// TIA Portal project "test" (V17)

(* hardware
DEVICE "S7-1500/ET200MP station_1"  S7-1500 station
   slot 0: "Rail_0"  Rack  6ES7 590-1***0-0AA0
   slot 1: "PLC_1"  CPU 1516-3 PN/DP  6ES7 516-3AN02-0AB0  V2.9
      slot 3: "CPU display_1"  6ES7591-1BA00-0AA0
      slot 32768: "PROFINET interface_1"  X1
      slot 33024: "PROFINET interface_2"  X2
      slot 33280: "DP interface_1"  X3
      slot 34817: "Virtual CP interface port_1"  Virtual CP interface port  Virtual CP interface port
DEVICE "S7-1500/ET200MP station_2"  S7-1500 station
   slot 0: "Rail_0"  Rack  6ES7 590-1***0-0AA0
   slot 1: "io device_1"  IM 155-5 PN HF  6ES7 155-5AA00-0AC0  V3.0
   slot 2: "DQ 32x24VDC/0.5A ST_1"  DQ 32x24VDC/0.5A ST  6ES7 522-1BL00-0AB0  V2.0
   slot 3: "AI 8xU/I/RTD/TC ST_1"  AI 8xU/I/RTD/TC ST  6ES7 531-7KF00-0AB0  V2.0
   slot 4: "AQ 4xU/I ST_1"  AQ 4xU/I ST  6ES7 532-5HD00-0AB0  V2.0
DEVICE "GSD device_1"  GSD.Device.PN
   slot 0: "Rack"  Rack  V1.0
   slot 0: "al1102_3"  AL1102  AL1102
      slot 0: "AL1102"  AL1102
      slot 1: "X1"  X1
         slot 1: "Port 1"  Port 1
         slot 2: "Port 2"  Port 2
      slot 1: "8 Ports_1"  8 Ports  AL1102
         slot 0: "IO-Link Master"  IO-Link Master
DEVICE "GSD device_2"  GSD.Device.PN
   slot 0: "Rack"  Rack  V1.0
   slot 0: "al1102_4"  AL1102  AL1102
      slot 0: "AL1102"  AL1102
      slot 1: "X1"  X1
         slot 1: "Port 1"  Port 1
         slot 2: "Port 2"  Port 2
      slot 1: "8 Ports_1"  8 Ports  AL1102
         slot 0: "IO-Link Master"  IO-Link Master
   slot 3: "IO-Link In  2 Byte + PQI"  IO-Link In  2 Byte + PQI
   slot 5: "IO-Link In  2 Byte + PQI_1"  IO-Link In  2 Byte + PQI
   slot 6: "IO-Link In  8 Byte + PQI"  IO-Link In  8 Byte + PQI
   slot 7: "IO-Link In  2 Byte + PQI_2"  IO-Link In  2 Byte + PQI
   slot 8: "IO-Link In  2 Byte + PQI_3"  IO-Link In  2 Byte + PQI
DEVICE "GSD device_3"  GSD.Device.PN
   slot 0: "Rack"  Rack  V1.0
   slot 0: "al1102_2"  AL1102  AL1102
      slot 0: "AL1102"  AL1102
      slot 1: "X1"  X1
         slot 1: "Port 1"  Port 1
         slot 2: "Port 2"  Port 2
      slot 1: "8 Ports_1"  8 Ports  AL1102
         slot 0: "IO-Link Master"  IO-Link Master
*)

// ===== PLC "PLC_1"  CPU 1516-3 PN/DP =====

VAR_GLOBAL   // PLC tag table "Default tag table"
   "firstHeater" AT %Q0.5 : Bool;
   "secondHeater" AT %Q0.6 : Bool;
   "thirdHeater" AT %Q0.7 : Bool;
   "tempAfter" AT %IW8 : Int;
   "tempBefore" AT %IW14 : Int;
   "valve" AT %QW8 : Int;
   "flowFlow" AT %IW32 : Int;
   "power" AT %MD50 : Real;
   "flowTemp" AT %IW34 : Int;
   "Tag_1" AT %M100.0 : Bool;
END_VAR

TYPE "UDT_Pomiar"
VERSION : 0.1
   STRUCT
      power : UDInt;
      switchesFirst : UDInt;
      switchesSecond : UDInt;
      switchesThird : UDInt;
      onePhase : UDInt;
      threePhase : UDInt;
   END_STRUCT;
END_TYPE

DATA_BLOCK "ExecutePWM_DB"   // DB1
{ S7_Optimized_Access := 'TRUE' }
VERSION : 0.1
// stored: InstanceOfName ExecutePWM
"ExecutePWM"
BEGIN
END_DATA_BLOCK

DATA_BLOCK "Analysis_DB"   // DB2
{ S7_Optimized_Access := 'TRUE' }
VERSION : 0.1
// stored: InstanceOfName Analysis
"Analysis"
BEGIN
END_DATA_BLOCK

// folder: System blocks/Program resources

DATA_BLOCK "IEC_Timer_0_DB_2"   // DB3
{ S7_Optimized_Access := 'TRUE' }
AUTHOR : Simatic
FAMILY : IEC
NAME : IEC_TMR
VERSION : 1.0
// stored: InstanceOfName IEC_TIMER
"IEC_TIMER"
BEGIN
END_DATA_BLOCK

DATA_BLOCK "IEC_Timer_0_DB_1"   // DB4
{ S7_Optimized_Access := 'TRUE' }
AUTHOR : Simatic
FAMILY : IEC
NAME : IEC_TMR
VERSION : 1.0
// stored: InstanceOfName IEC_TIMER
"IEC_TIMER"
BEGIN
END_DATA_BLOCK

// folder: (top level)

FUNCTION_BLOCK "ControlPWM"   // FB1, LAD
TITLE = ControlPWM
{ S7_Optimized_Access := 'TRUE' }
VERSION : 0.1
// Obsługa wypełnienia dla każdej z grzałek, w zależności od wyboru trybu pracy (jednofazowy lub trójfazowy).
   VAR_INPUT
      I_cycleTime : DInt;   // given in milliseconds
      I_filling_1 : Int;   // <0, 100>
      I_filling_2 : Int;   // <0, 100>
      I_filling_3 : Int;   // <0, 100>
      I_OnePhaseSwitch : Bool;
      I_threePhaseSwitch : Bool;
   END_VAR
   VAR_OUTPUT
      O_heaterState_1 : Bool;
      O_heaterState_2 : Bool;
      O_heaterState_3 : Bool;
   END_VAR
   VAR
      IEC_Timer_11 : TON_TIME;
      IEC_Timer_12 : TON_TIME;
      highStateNum_1 : DInt;   // given in milliseconds
      lowStateNum_1 : DInt;   // given in milliseconds
      highStateTime_1 : Time;   // given in milliseconds
      lowStateTime_1 : Time;   // given in milliseconds
      IEC_Timer_21 : TON_TIME;
      IEC_Timer_22 : TON_TIME;
      highStateNum_2 : DInt;   // given in milliseconds
      lowStateNum_2 : DInt;   // given in milliseconds
      highStateTime_2 : Time;   // given in milliseconds
      lowStateTime_2 : Time;   // given in milliseconds
      IEC_Timer_31 : TON_TIME;
      IEC_Timer_32 : TON_TIME;
      highStateNum_3 : DInt;   // given in milliseconds
      lowStateNum_3 : DInt;   // given in milliseconds
      highStateTime_3 : Time;   // given in milliseconds
      lowStateTime_3 : Time;   // given in milliseconds
      IEC_Timer_0_Instance : TON_TIME;
      IEC_Timer_0_Instance_1 : TON_TIME;
   END_VAR
BEGIN

REGION Network 1: Obliczenie czasu stanów
   // Blok calculate oblicza czas na podstawie wartości procentowej (I_filling_X) i przypisuje wartości czasowe stanu wysokiego oraz niskiego (Int) do odpowiednich zmiennych (highStateNum_X, lowStateNum_X).
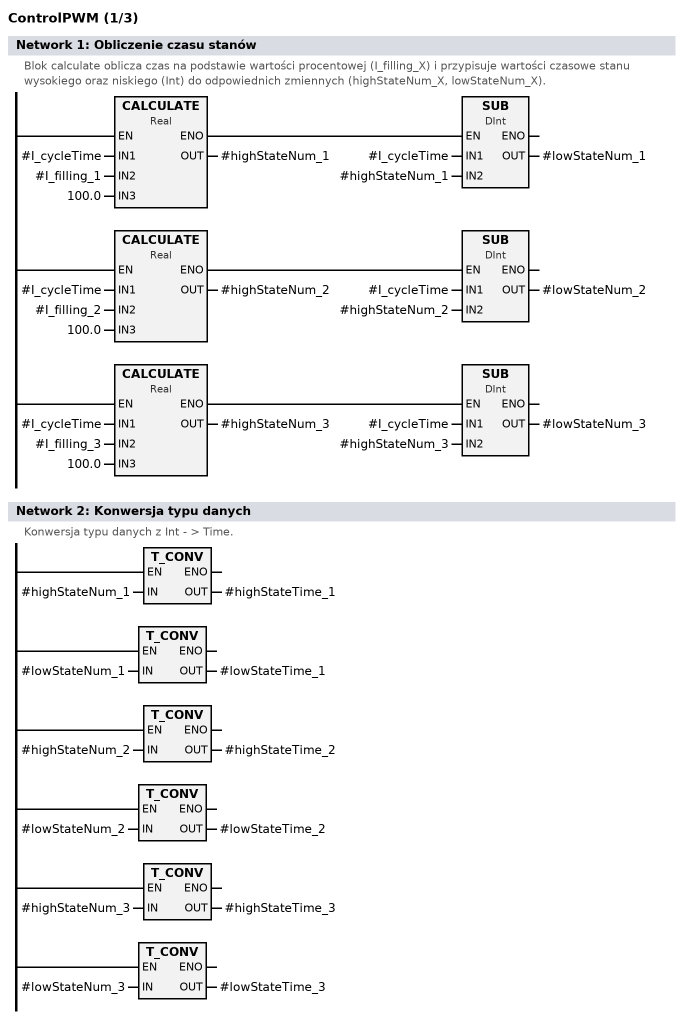
   RUNG wire#powerrail
      { S7_Templates := "SrcType := Real"; S7_Expression := "(IN1*IN2)/IN3" } Calculate(in1 := #I_cycleTime, in2 := #I_filling_1, in3 := 100.0, out => #highStateNum_1)
      { S7_Templates := "SrcType := DInt" } Sub(in1 := #I_cycleTime, in2 := #highStateNum_1, out => #lowStateNum_1)
   END_RUNG
   RUNG wire#powerrail
      { S7_Templates := "SrcType := Real"; S7_Expression := "(IN1*IN2)/IN3" } Calculate(in1 := #I_cycleTime, in2 := #I_filling_2, in3 := 100.0, out => #highStateNum_2)
      { S7_Templates := "SrcType := DInt" } Sub(in1 := #I_cycleTime, in2 := #highStateNum_2, out => #lowStateNum_2)
   END_RUNG
   RUNG wire#powerrail
      { S7_Templates := "SrcType := Real"; S7_Expression := "(IN1*IN2)/IN3" } Calculate(in1 := #I_cycleTime, in2 := #I_filling_3, in3 := 100.0, out => #highStateNum_3)
      { S7_Templates := "SrcType := DInt" } Sub(in1 := #I_cycleTime, in2 := #highStateNum_3, out => #lowStateNum_3)
   END_RUNG
   // the same network as SCL:
   #highStateNum_1 := (#I_cycleTime*#I_filling_1)/100.0;
   #lowStateNum_1 := #I_cycleTime - #highStateNum_1;
   #highStateNum_2 := (#I_cycleTime*#I_filling_2)/100.0;
   #lowStateNum_2 := #I_cycleTime - #highStateNum_2;
   #highStateNum_3 := (#I_cycleTime*#I_filling_3)/100.0;
   #lowStateNum_3 := #I_cycleTime - #highStateNum_3;
END_REGION

REGION Network 2: Konwersja typu danych
   // Konwersja typu danych z Int - > Time.
   #highStateTime_1 := T_CONV(IN := #highStateNum_1);
   #lowStateTime_1 := T_CONV(IN := #lowStateNum_1);
   #highStateTime_2 := T_CONV(IN := #highStateNum_2);
   #lowStateTime_2 := T_CONV(IN := #lowStateNum_2);
   #highStateTime_3 := T_CONV(IN := #highStateNum_3);
   #lowStateTime_3 := T_CONV(IN := #lowStateNum_3);
END_REGION

REGION Network 3: Kontrola wypełnienia trybu trójfazowego (1)
   // Wypełnienie jest kontrolowane na podstawie dwóch zegarów TON. Każdy ze stanów uruchamia zegar, który odlicza czas (opóźninie) do uruchomienia stanu przeciwnego. Timery działają na przemian i nie mogą zostac uruchomione jednocześnie. Po zmianie stanu, licznik stanu przeciwnego zostaje zresetowany zgodnie z działaniem zegara TON. Logika ta działa nieprawidłowo, gdy któryś z określonych czasów jest równy 0, stąd dwie ostatnie gałęzie usprawniające działanie.
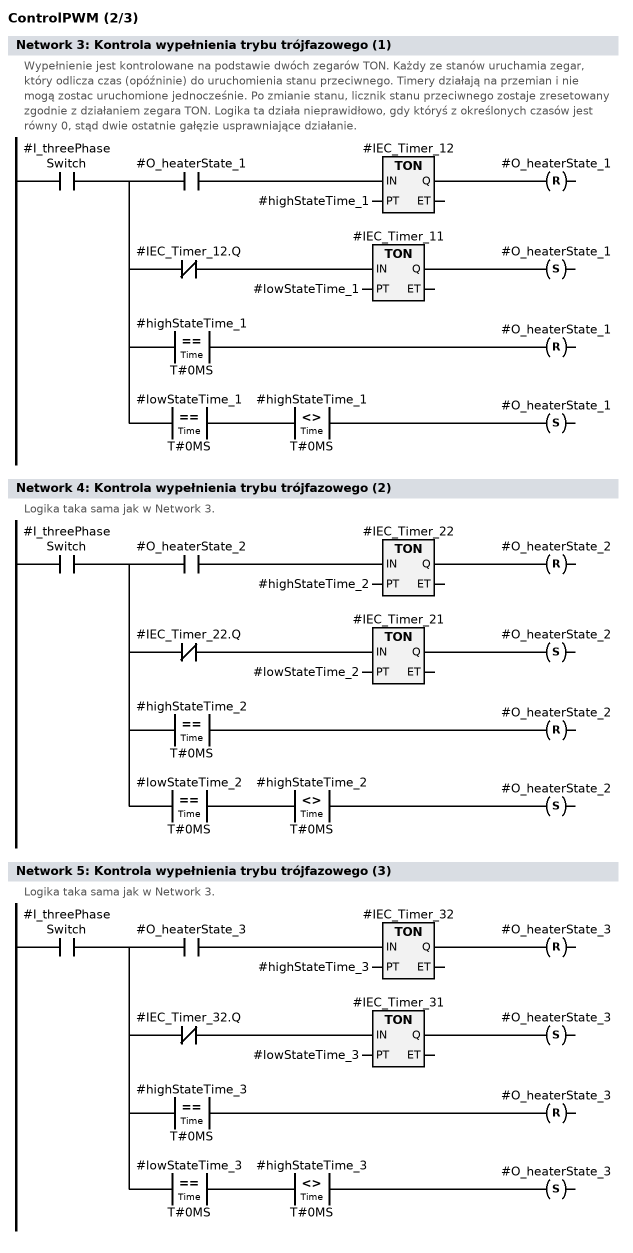
   #IEC_Timer_12(IN := #I_threePhaseSwitch AND #O_heaterState_1, PT := #highStateTime_1);   // TON
   IF #IEC_Timer_12.Q THEN #O_heaterState_1 := FALSE; END_IF;
   #IEC_Timer_11(IN := #I_threePhaseSwitch AND NOT #IEC_Timer_12.Q, PT := #lowStateTime_1);   // TON
   IF #IEC_Timer_11.Q THEN #O_heaterState_1 := TRUE; END_IF;
   IF #I_threePhaseSwitch AND (#highStateTime_1 = T#0MS) THEN #O_heaterState_1 := FALSE; END_IF;
   IF #I_threePhaseSwitch AND (#lowStateTime_1 = T#0MS) AND (#highStateTime_1 <> T#0MS) THEN
       #O_heaterState_1 := TRUE;
   END_IF;
END_REGION

REGION Network 4: Kontrola wypełnienia trybu trójfazowego (2)
   // Logika taka sama jak w Network 3.
   #IEC_Timer_22(IN := #I_threePhaseSwitch AND #O_heaterState_2, PT := #highStateTime_2);   // TON
   IF #IEC_Timer_22.Q THEN #O_heaterState_2 := FALSE; END_IF;
   #IEC_Timer_21(IN := #I_threePhaseSwitch AND NOT #IEC_Timer_22.Q, PT := #lowStateTime_2);   // TON
   IF #IEC_Timer_21.Q THEN #O_heaterState_2 := TRUE; END_IF;
   IF #I_threePhaseSwitch AND (#highStateTime_2 = T#0MS) THEN #O_heaterState_2 := FALSE; END_IF;
   IF #I_threePhaseSwitch AND (#lowStateTime_2 = T#0MS) AND (#highStateTime_2 <> T#0MS) THEN
       #O_heaterState_2 := TRUE;
   END_IF;
END_REGION

REGION Network 5: Kontrola wypełnienia trybu trójfazowego (3)
   // Logika taka sama jak w Network 3.
   #IEC_Timer_32(IN := #I_threePhaseSwitch AND #O_heaterState_3, PT := #highStateTime_3);   // TON
   IF #IEC_Timer_32.Q THEN #O_heaterState_3 := FALSE; END_IF;
   #IEC_Timer_31(IN := #I_threePhaseSwitch AND NOT #IEC_Timer_32.Q, PT := #lowStateTime_3);   // TON
   IF #IEC_Timer_31.Q THEN #O_heaterState_3 := TRUE; END_IF;
   IF #I_threePhaseSwitch AND (#highStateTime_3 = T#0MS) THEN #O_heaterState_3 := FALSE; END_IF;
   IF #I_threePhaseSwitch AND (#lowStateTime_3 = T#0MS) AND (#highStateTime_3 <> T#0MS) THEN
       #O_heaterState_3 := TRUE;
   END_IF;
END_REGION

REGION Network 6: Kontrola wypełnienia trybu jednofazowego
   // Logika taka sama jak w przypadku trybu trójfazowego, ale wszystkie trzy grzałki w danej chwili czasu mają taki sam stan.
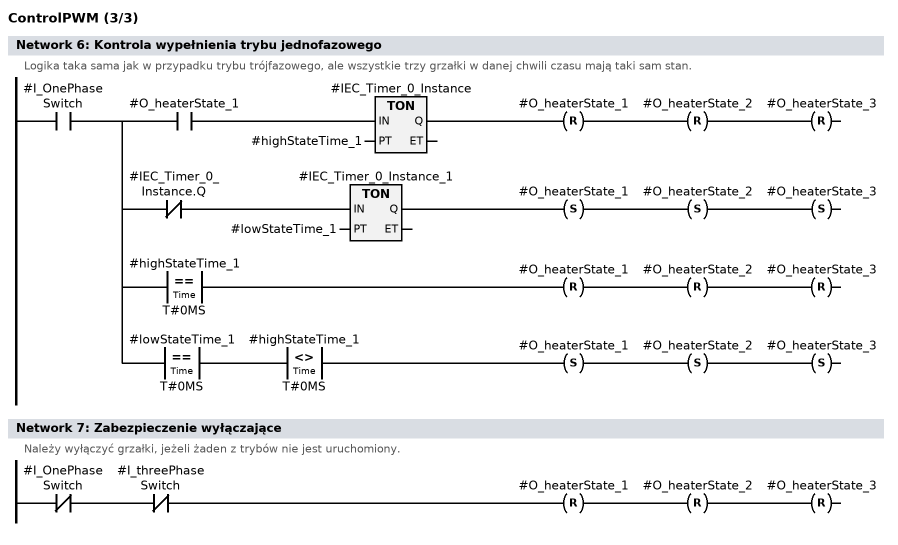
   #IEC_Timer_0_Instance(IN := #I_OnePhaseSwitch AND #O_heaterState_1, PT := #highStateTime_1);   // TON
   IF #IEC_Timer_0_Instance.Q THEN
       #O_heaterState_1 := FALSE;
       #O_heaterState_2 := FALSE;
       #O_heaterState_3 := FALSE;
   END_IF;
   #IEC_Timer_0_Instance_1(IN := #I_OnePhaseSwitch AND NOT #IEC_Timer_0_Instance.Q, PT := #lowStateTime_1);   // TON
   IF #IEC_Timer_0_Instance_1.Q THEN
       #O_heaterState_1 := TRUE;
       #O_heaterState_2 := TRUE;
       #O_heaterState_3 := TRUE;
   END_IF;
   IF #I_OnePhaseSwitch AND (#highStateTime_1 = T#0MS) THEN
       #O_heaterState_1 := FALSE;
       #O_heaterState_2 := FALSE;
       #O_heaterState_3 := FALSE;
   END_IF;
   IF #I_OnePhaseSwitch AND (#lowStateTime_1 = T#0MS) AND (#highStateTime_1 <> T#0MS) THEN
       #O_heaterState_1 := TRUE;
       #O_heaterState_2 := TRUE;
       #O_heaterState_3 := TRUE;
   END_IF;
END_REGION

REGION Network 7: Zabezpieczenie wyłączające
   // Należy wyłączyć grzałki, jeżeli żaden z trybów nie jest uruchomiony.
   RUNG wire#powerrail
      I_Contact( #I_OnePhaseSwitch )
      I_Contact( #I_threePhaseSwitch )
      R_Coil( #O_heaterState_1 )
      R_Coil( #O_heaterState_2 )
      R_Coil( #O_heaterState_3 )
   END_RUNG
   // the same network as SCL:
   IF NOT #I_OnePhaseSwitch AND NOT #I_threePhaseSwitch THEN
       #O_heaterState_1 := FALSE;
       #O_heaterState_2 := FALSE;
       #O_heaterState_3 := FALSE;
   END_IF;
END_REGION
END_FUNCTION_BLOCK

FUNCTION_BLOCK "ExecutePWM"   // FB2, LAD
TITLE = ExecutePWM
{ S7_Optimized_Access := 'TRUE' }
VERSION : 0.1
// Określenie potrzebnych parametrów oraz fizyczne obiciążenie każdej z grzałek.
   VAR_INPUT
      I_flowSetPoint : Real;
      I_tempSetPoint : Real;
      I_furnancePower : Real := 0.0;
      I_switchTime_s : Real := 30.0;   // given in seconds
      I_cycleTime_s : Real := 1.0;   // given in seconds
   END_VAR
   VAR_OUTPUT
      O_firstState : Bool;
      O_secondState : Bool;
      O_thirdState : Bool;
   END_VAR
   VAR_IN_OUT
      IO_onePhaseSwitch : Bool;
      IO_threePhaseSwitch : Bool;
   END_VAR
   VAR
      tempAfterScaled : Real;
      tempAfterNormalised : Real;
      flowTemp : Real;
      flowFlow : Real;
      tempOK : Bool := false;
      flowOK : Bool := false;
      ControlPWM_Instance : "ControlPWM";
      cycleTime_ms : DInt;   // given in milliseconds
      switchTime_ms : DInt;
      switchTime : Time;
      firstHeater : Int;
      secondHeater : Int;
      thirdHeater : Int;
      enablePWM : Bool;
      cycleCount : Int;
      fullCycleTimer : TON_TIME;
      pulseInc : TP_TIME;
      pulseTrigger : Bool;
      firstFilling : Real;
      secondFilling : Real;
      thirdFilling : Real;
      heaterFactor : Real;
      onePhaseActive : Bool;
      threePhaseActive : Bool;
      ControlPWM_Instance_1 : "ControlPWM";
   END_VAR
   VAR CONSTANT
      C_numberOfHeaters : Real := 3.0;
   END_VAR
   VAR_TEMP   // added for the SCL form of the ladder/FBD networks
      _w1 : Bool;
      _w2 : Bool;
   END_VAR
BEGIN

REGION Network 1: Kontrola wyboru trybu
   // W jednej chwili może być aktywny tylko jeden z trybów pracy. Włączenie jednego trybu dezaktywuje drugi.
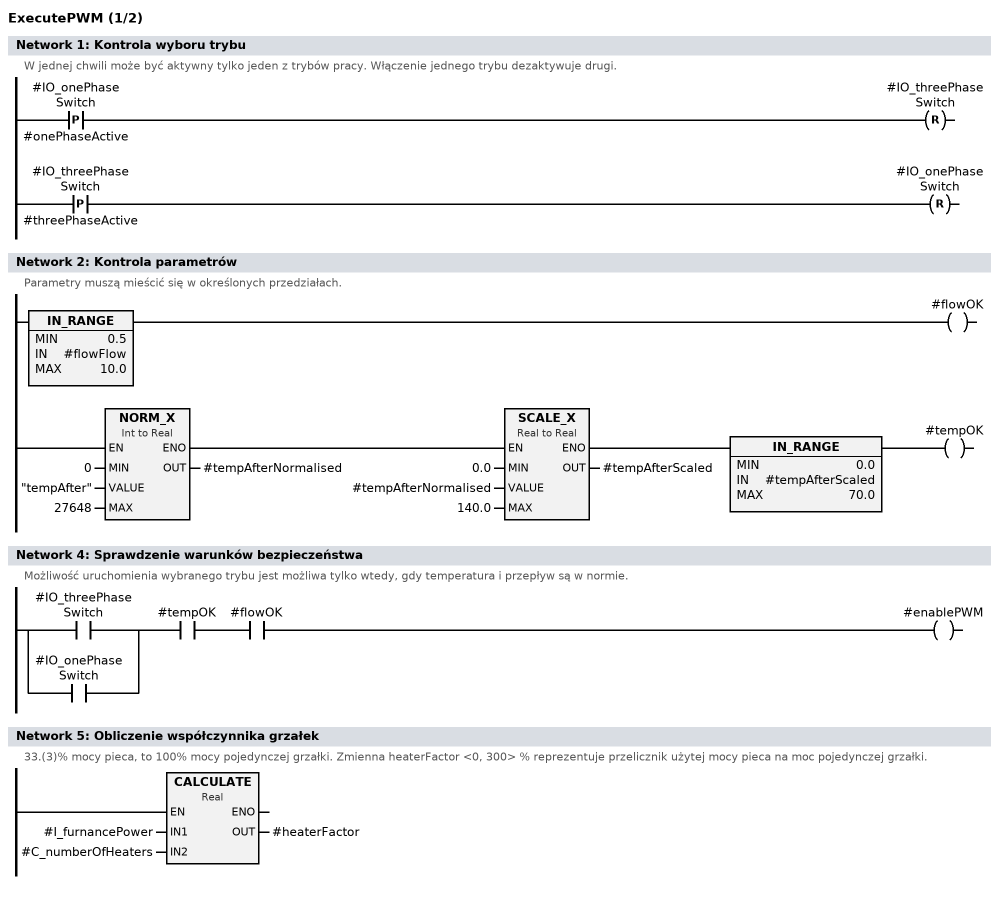
   RUNG wire#powerrail
      P_Contact(operand := #IO_onePhaseSwitch, bit := #onePhaseActive)
      R_Coil( #IO_threePhaseSwitch )
   END_RUNG
   RUNG wire#powerrail
      P_Contact(operand := #IO_threePhaseSwitch, bit := #threePhaseActive)
      R_Coil( #IO_onePhaseSwitch )
   END_RUNG
   // the same network as SCL:
   #_w1 := #IO_onePhaseSwitch AND NOT #onePhaseActive;   // rising edge of #IO_onePhaseSwitch
   #onePhaseActive := #IO_onePhaseSwitch;
   IF #_w1 THEN #IO_threePhaseSwitch := FALSE; END_IF;
   #_w2 := #IO_threePhaseSwitch AND NOT #threePhaseActive;   // rising edge of #IO_threePhaseSwitch
   #threePhaseActive := #IO_threePhaseSwitch;
   IF #_w2 THEN #IO_onePhaseSwitch := FALSE; END_IF;
END_REGION

REGION Network 2: Kontrola parametrów
   // Parametry muszą mieścić się w określonych przedziałach.
   RUNG wire#powerrail
      { S7_Templates := "SrcType := Real" } InRange(min := 0.5, in := #flowFlow, max := 10.0)
      Coil( #flowOK )
   END_RUNG
   RUNG wire#powerrail
      { S7_Templates := "[SrcType := Int, DestType := Real]" } Normalize(min := 0, value := "tempAfter", max := 27648, out => #tempAfterNormalised)
      { S7_Templates := "[SrcType := Real, DestType := Real]" } Scale(min := 0.0, value := #tempAfterNormalised, max := 140.0, out => #tempAfterScaled)
      { S7_Templates := "SrcType := Real" } InRange(min := 0.0, in := #tempAfterScaled, max := 70.0)
      Coil( #tempOK )
   END_RUNG
   // the same network as SCL:
   #flowOK := (0.5 <= #flowFlow) AND (#flowFlow <= 10.0);
   #tempAfterNormalised := NORM_X(MIN := 0, VALUE := "tempAfter", MAX := 27648);
   #tempAfterScaled := SCALE_X(MIN := 0.0, VALUE := #tempAfterNormalised, MAX := 140.0);
   #tempOK := (0.0 <= #tempAfterScaled) AND (#tempAfterScaled <= 70.0);
END_REGION

REGION Network 3 (SCL): Parametry
   #flowFlow := INT_TO_REAL(WORD_TO_INT("flowFlow")) * 0.01;
   #flowTemp := INT_TO_REAL(WORD_TO_INT("flowTemp")) * 0.1;
END_REGION

REGION Network 4: Sprawdzenie warunków bezpieczeństwa
   // Możliwość uruchomienia wybranego trybu jest możliwa tylko wtedy, gdy temperatura i przepływ są w normie.
   RUNG wire#powerrail
      Contact( #IO_threePhaseSwitch )
      wire#w1
      Contact( #tempOK )
      Contact( #flowOK )
      Coil( #enablePWM )
   END_RUNG
   RUNG wire#powerrail
      Contact( #IO_onePhaseSwitch )
   END_RUNG wire#w1
   // the same network as SCL:
   #enablePWM := (#IO_threePhaseSwitch OR #IO_onePhaseSwitch) AND #tempOK AND #flowOK;
END_REGION

REGION Network 5: Obliczenie współczynnika grzałek
   // 33.(3)% mocy pieca, to 100% mocy pojedynczej grzałki. Zmienna heaterFactor <0, 300> % reprezentuje przelicznik użytej mocy pieca na moc pojedynczej grzałki.
   RUNG wire#powerrail
      { S7_Templates := "SrcType := Real"; S7_Expression := "(IN1 * IN2)" } Calculate(in1 := #I_furnancePower, in2 := #C_numberOfHeaters, out => #heaterFactor)
   END_RUNG
   // the same network as SCL:
   #heaterFactor := (#I_furnancePower * #C_numberOfHeaters);
END_REGION

REGION Network 6: Obliczenie współczynników wypełnienia dla trybu trójfazowego
   // Na podstawie zmiennej heaterFactor, wypełnienia zostają rozdystrybuowane pomiędzy poszczególne grzałki. Każda z kolejnych grzałek otrzymuje maksymalne możliwe obciążenie <0,100> % (zmienne first/second/thirdFilling).
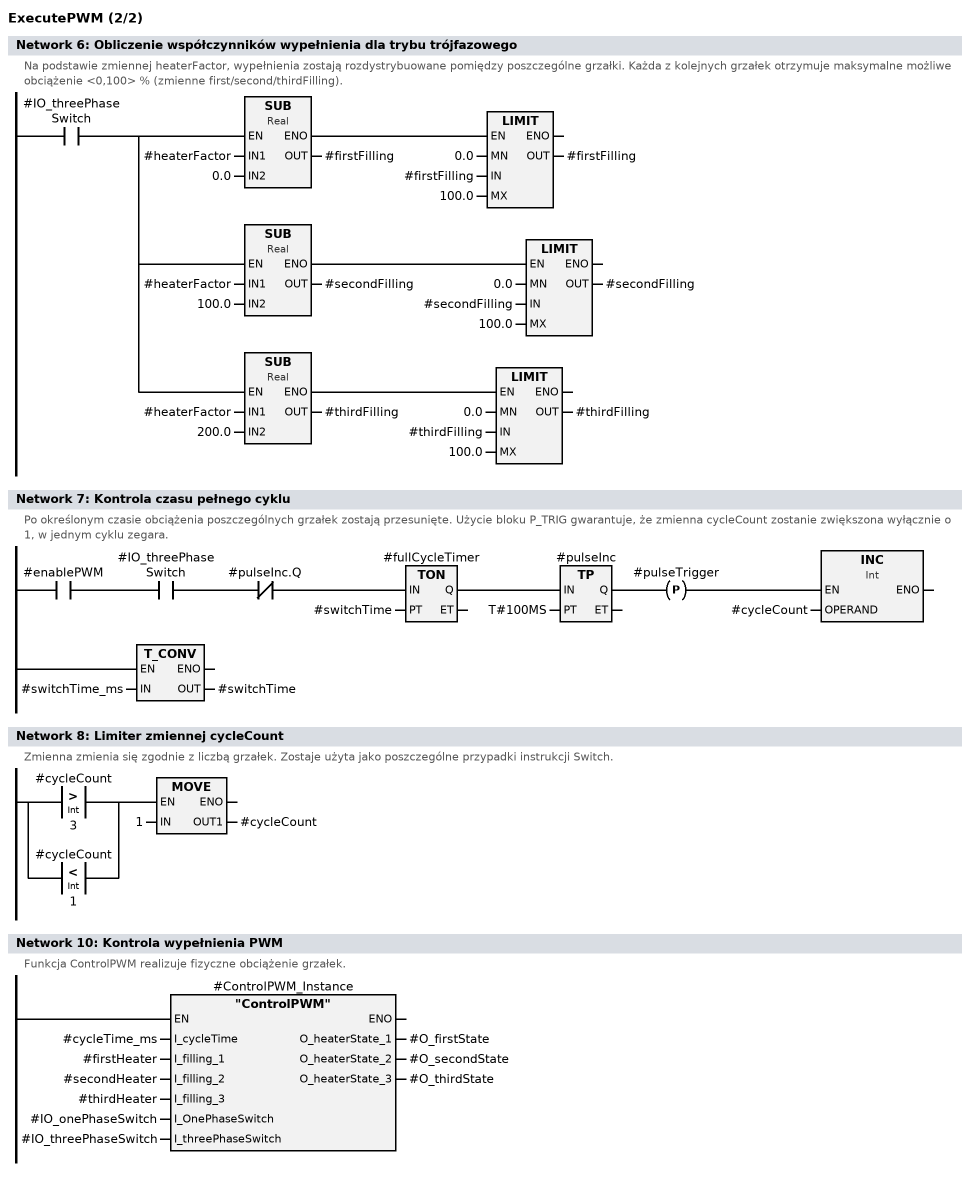
   IF #IO_threePhaseSwitch THEN
       #firstFilling := #heaterFactor - 0.0;
       #firstFilling := LIMIT(MN := 0.0, IN := #firstFilling, MX := 100.0);
       #secondFilling := #heaterFactor - 100.0;
       #secondFilling := LIMIT(MN := 0.0, IN := #secondFilling, MX := 100.0);
       #thirdFilling := #heaterFactor - 200.0;
       #thirdFilling := LIMIT(MN := 0.0, IN := #thirdFilling, MX := 100.0);
   END_IF;
END_REGION

REGION Network 7: Kontrola czasu pełnego cyklu
   // Po określonym czasie obciążenia poszczególnych grzałek zostają przesunięte. Użycie bloku P_TRIG gwarantuje, że zmienna cycleCount zostanie zwiększona wyłącznie o 1, w jednym cyklu zegara.
   #fullCycleTimer(IN := #enablePWM AND #IO_threePhaseSwitch AND NOT #pulseInc.Q, PT := #switchTime);   // TON
   #pulseInc(IN := #fullCycleTimer.Q, PT := T#100MS);   // TP
   #_w1 := #pulseInc.Q AND NOT #pulseTrigger;   // rising edge
   #pulseTrigger := #pulseInc.Q;
   IF #_w1 THEN #cycleCount := #cycleCount + 1; END_IF;
   #switchTime := T_CONV(IN := #switchTime_ms);
END_REGION

REGION Network 8: Limiter zmiennej cycleCount
   // Zmienna zmienia się zgodnie z liczbą grzałek. Zostaje użyta jako poszczególne przypadki instrukcji Switch.
   RUNG wire#powerrail
      { S7_Templates := "SrcType := Int" } GT_Contact(in1 := #cycleCount, in2 := 3)
      wire#w1
      Move(in := 1, out1 => #cycleCount)
   END_RUNG
   RUNG wire#powerrail
      { S7_Templates := "SrcType := Int" } LT_Contact(in1 := #cycleCount, in2 := 1)
   END_RUNG wire#w1
   // the same network as SCL:
   IF (#cycleCount > 3) OR (#cycleCount < 1) THEN #cycleCount := 1; END_IF;
END_REGION

REGION Network 9 (SCL): Obciążanie w zależności od cyklu
   // Po określonym czasie cyklu, zmienna cycleCount zwiększa się. W zależności od jej wartości wybrany zostaje jeden z trzech przypadków obciążenia grzałek, dla trybu trójfazowego. Dla trybu jednofazowego każda z grzałek zostaje obciążona równomiernie, wartością użytej aktualnie mocy pieca.
   #cycleTime_ms := REAL_TO_DINT(#I_cycleTime_s * 1000);
   #switchTime_ms := REAL_TO_DINT(#I_switchTime_s * 1000);

   IF #IO_threePhaseSwitch THEN
       CASE #cycleCount OF
           1:  
               #firstHeater := REAL_TO_INT(#firstFilling);
               #secondHeater := REAL_TO_INT(#secondFilling);
               #thirdHeater := REAL_TO_INT(#thirdFilling);
           2:  
               #firstHeater := REAL_TO_INT(#thirdFilling);
               #secondHeater := REAL_TO_INT(#firstFilling);
               #thirdHeater := REAL_TO_INT(#secondFilling);
           3:
               #firstHeater := REAL_TO_INT(#secondFilling);
               #secondHeater := REAL_TO_INT(#thirdFilling);
               #thirdHeater := REAL_TO_INT(#firstFilling);
       END_CASE;
   END_IF;

   IF #IO_onePhaseSwitch THEN
       #firstHeater := REAL_TO_INT(#I_furnancePower);
       #secondHeater := REAL_TO_INT(#I_furnancePower);
       #thirdHeater := REAL_TO_INT(#I_furnancePower);
   END_IF;

   IF #enablePWM = false THEN
       #firstHeater := 0;
       #secondHeater := 0;
       #thirdHeater := 0;
   END_IF;
END_REGION

REGION Network 10: Kontrola wypełnienia PWM
   // Funkcja ControlPWM realizuje fizyczne obciążenie grzałek.
   RUNG wire#powerrail
      #ControlPWM_Instance(I_cycleTime := #cycleTime_ms, I_filling_1 := #firstHeater, I_filling_2 := #secondHeater, I_filling_3 := #thirdHeater, I_OnePhaseSwitch := #IO_onePhaseSwitch, I_threePhaseSwitch := #IO_threePhaseSwitch, O_heaterState_1 => #O_firstState, O_heaterState_2 => #O_secondState, O_heaterState_3 => #O_thirdState)
   END_RUNG
   // the same network as SCL:
   #ControlPWM_Instance(I_cycleTime := #cycleTime_ms,   // "ControlPWM"
                        I_filling_1 := #firstHeater,
                        I_filling_2 := #secondHeater,
                        I_filling_3 := #thirdHeater,
                        I_OnePhaseSwitch := #IO_onePhaseSwitch,
                        I_threePhaseSwitch := #IO_threePhaseSwitch,
                        O_heaterState_1 => #O_firstState,
                        O_heaterState_2 => #O_secondState,
                        O_heaterState_3 => #O_thirdState);
END_REGION
END_FUNCTION_BLOCK

FUNCTION_BLOCK "Analysis"   // FB3, LAD
TITLE = Analysis
{ S7_Optimized_Access := 'TRUE' }
VERSION : 0.1
// Automatyczne zmienianie parametrów i zapis w celu analizy danych.
   VAR_INPUT
      I_first : Bool;
      I_second : Bool;
      I_third : Bool;
      I_switchTime : DInt;
      I_reset : Bool;
      I_start : Bool;
   END_VAR
   VAR_IN_OUT
      IO_power : Real;
      IO_onePhase : Bool;
      IO_threePhase : Bool;
   END_VAR
   VAR
      switchesFirst : UDInt;
      switchesSecond : UDInt;
      switchesThird : UDInt;
      I_first_NT : Bool;
      I_first_PT : Bool;
      I_second_NT : Bool;
      I_second_PT : Bool;
      I_third_NT : Bool;
      I_third_PT : Bool;
      whichCase : Int;
      caseTime : Time;
      IEC_Timer_0_Instance : TON_TIME;
      IEC_Timer_0_Instance_1 : TP_TIME;
      case_PT : Bool;
      DATA : Array[0..7] of "UDT_Pomiar";
   END_VAR
   VAR_TEMP   // added for the SCL form of the ladder/FBD networks
      _w1 : Bool;
      _w2 : Bool;
      _w3 : Bool;
      _w4 : Bool;
      _w5 : Bool;
      _w6 : Bool;
   END_VAR
BEGIN

REGION Network 1: Ustawianie bazowe
   // ...
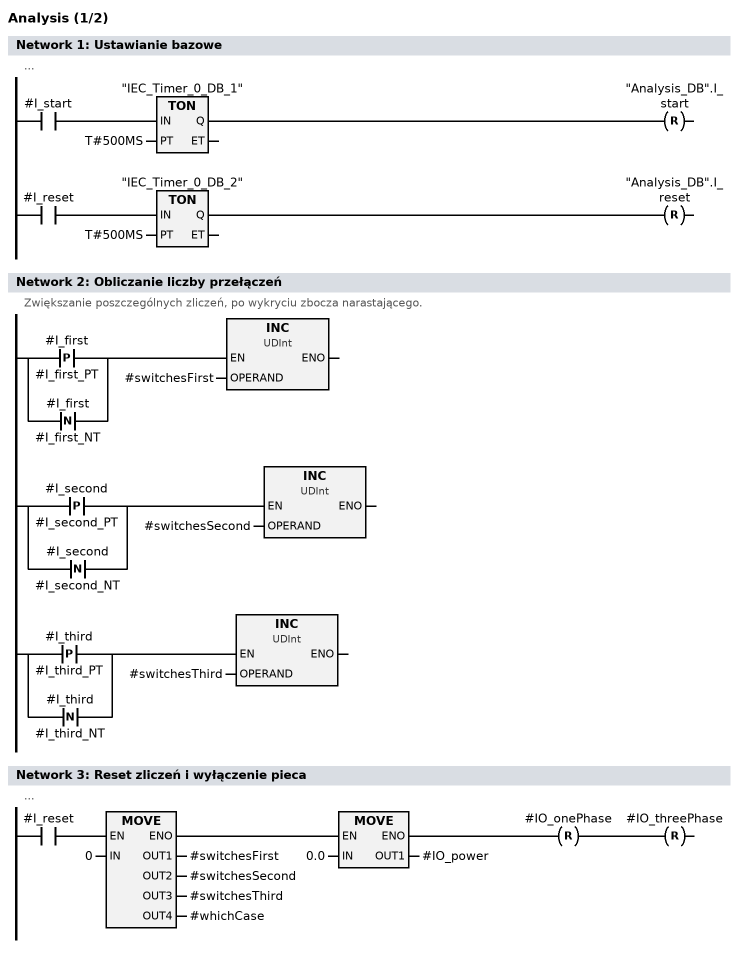
   "IEC_Timer_0_DB_1".TON(IN := #I_start, PT := T#500MS);
   IF "IEC_Timer_0_DB_1".Q THEN "Analysis_DB".I_start := FALSE; END_IF;
   "IEC_Timer_0_DB_2".TON(IN := #I_reset, PT := T#500MS);
   IF "IEC_Timer_0_DB_2".Q THEN "Analysis_DB".I_reset := FALSE; END_IF;
END_REGION

REGION Network 2: Obliczanie liczby przełączeń
   // Zwiększanie poszczególnych zliczeń, po wykryciu zbocza narastającego.
   RUNG wire#powerrail
      P_Contact(operand := #I_first, bit := #I_first_PT)
      wire#w1
      { S7_Templates := "DestType := UDInt" } Inc( #switchesFirst )
   END_RUNG
   RUNG wire#powerrail
      N_Contact(operand := #I_first, bit := #I_first_NT)
   END_RUNG wire#w1
   RUNG wire#powerrail
      P_Contact(operand := #I_second, bit := #I_second_PT)
      wire#w2
      { S7_Templates := "DestType := UDInt" } Inc( #switchesSecond )
   END_RUNG
   RUNG wire#powerrail
      N_Contact(operand := #I_second, bit := #I_second_NT)
   END_RUNG wire#w2
   RUNG wire#powerrail
      P_Contact(operand := #I_third, bit := #I_third_PT)
      wire#w3
      { S7_Templates := "DestType := UDInt" } Inc( #switchesThird )
   END_RUNG
   RUNG wire#powerrail
      N_Contact(operand := #I_third, bit := #I_third_NT)
   END_RUNG wire#w3
   // the same network as SCL:
   #_w1 := #I_first AND NOT #I_first_PT;   // rising edge of #I_first
   #I_first_PT := #I_first;
   #_w2 := NOT #I_first AND #I_first_NT;   // falling edge of #I_first
   #I_first_NT := #I_first;
   IF #_w1 OR #_w2 THEN #switchesFirst := #switchesFirst + 1; END_IF;
   #_w3 := #I_second AND NOT #I_second_PT;   // rising edge of #I_second
   #I_second_PT := #I_second;
   #_w4 := NOT #I_second AND #I_second_NT;   // falling edge of #I_second
   #I_second_NT := #I_second;
   IF #_w3 OR #_w4 THEN #switchesSecond := #switchesSecond + 1; END_IF;
   #_w5 := #I_third AND NOT #I_third_PT;   // rising edge of #I_third
   #I_third_PT := #I_third;
   #_w6 := NOT #I_third AND #I_third_NT;   // falling edge of #I_third
   #I_third_NT := #I_third;
   IF #_w5 OR #_w6 THEN #switchesThird := #switchesThird + 1; END_IF;
END_REGION

REGION Network 3: Reset zliczeń i wyłączenie pieca
   // ...
   RUNG wire#powerrail
      Contact( #I_reset )
      Move(in := 0, out1 => #switchesFirst, out2 => #switchesSecond, out3 => #switchesThird, out4 => #whichCase)
      Move(in := 0.0, out1 => #IO_power)
      R_Coil( #IO_onePhase )
      R_Coil( #IO_threePhase )
   END_RUNG
   // the same network as SCL:
   IF #I_reset THEN
       #switchesFirst := 0;
       #switchesSecond := 0;
       #switchesThird := 0;
       #whichCase := 0;
       #IO_power := 0.0;
       #IO_onePhase := FALSE;
       #IO_threePhase := FALSE;
   END_IF;
END_REGION

REGION Network 4: Zapis informajci w tabelach.
   // Dane są zapisywane w tabelach w określonej kolejności:
   // 1. moc pieca
   // 2. przełączenia pierwszej grzałki
   // 3. przełączenia drugiej grzałki
   // 4. przełączenia trzeciej grzałki
   // 5. tryb jednofazowy (true/false, 1/0)
   // 6. tryb trójfazowy (true/false, 1/0)
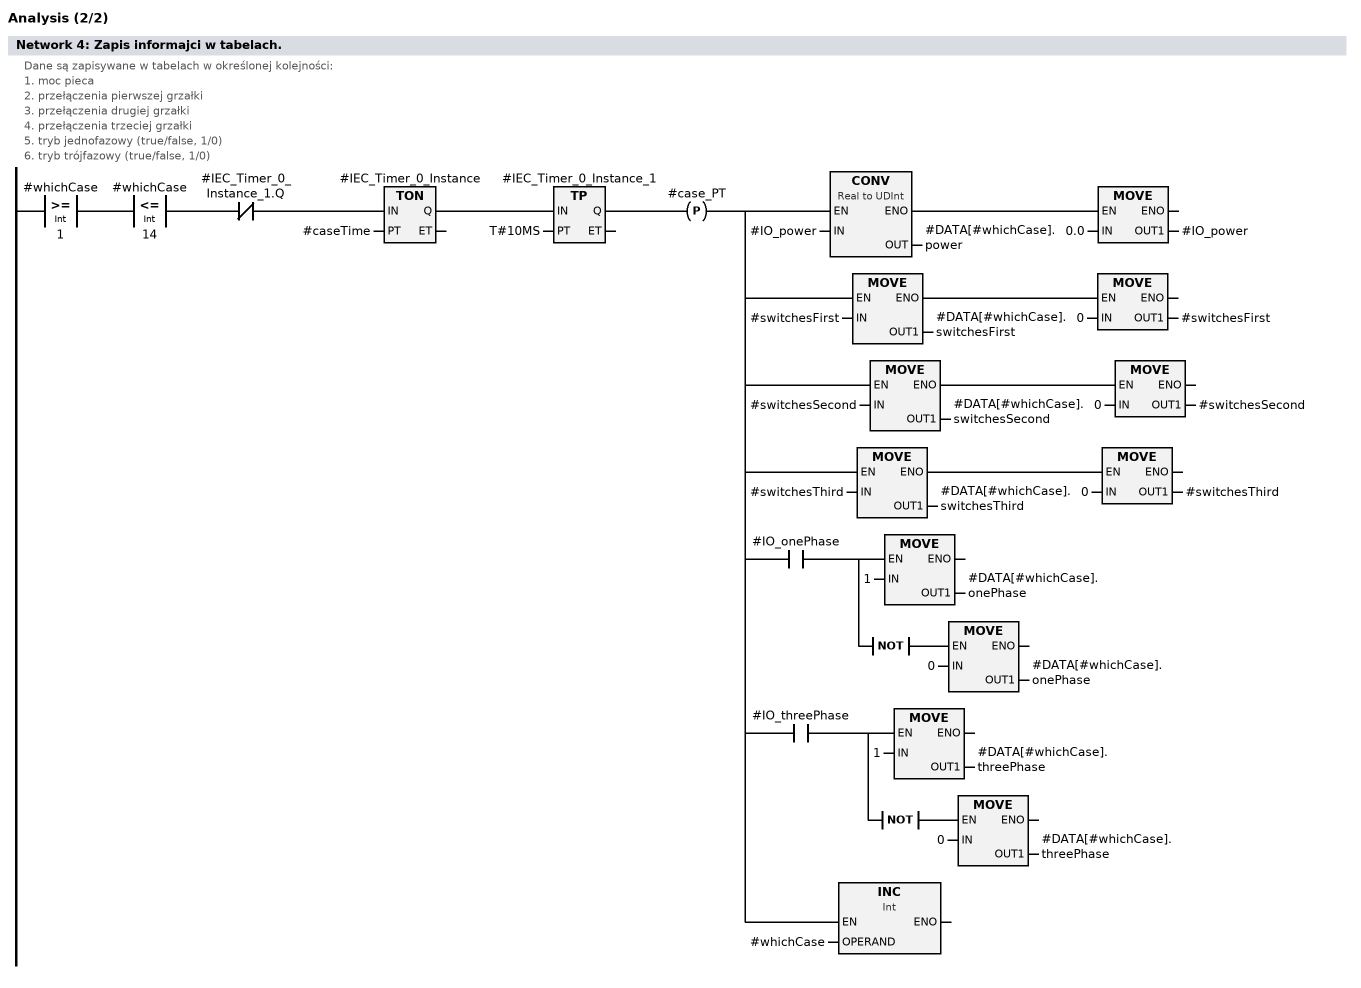
   #IEC_Timer_0_Instance(IN := (#whichCase >= 1) AND (#whichCase <= 14) AND NOT #IEC_Timer_0_Instance_1.Q,   // TON
                         PT := #caseTime);
   #IEC_Timer_0_Instance_1(IN := #IEC_Timer_0_Instance.Q, PT := T#10MS);   // TP
   #_w1 := #IEC_Timer_0_Instance_1.Q AND NOT #case_PT;   // rising edge
   #case_PT := #IEC_Timer_0_Instance_1.Q;
   IF #_w1 THEN
       #DATA[#whichCase].power := REAL_TO_UDINT(#IO_power);
       #IO_power := 0.0;
       #DATA[#whichCase].switchesFirst := #switchesFirst;
       #switchesFirst := 0;
       #DATA[#whichCase].switchesSecond := #switchesSecond;
       #switchesSecond := 0;
       #DATA[#whichCase].switchesThird := #switchesThird;
       #switchesThird := 0;
   END_IF;
   #_w2 := #_w1 AND #IO_onePhase;
   IF #_w2 THEN #DATA[#whichCase].onePhase := 1; END_IF;
   IF NOT #_w2 THEN #DATA[#whichCase].onePhase := 0; END_IF;
   #_w3 := #_w1 AND #IO_threePhase;
   IF #_w3 THEN #DATA[#whichCase].threePhase := 1; END_IF;
   IF NOT #_w3 THEN #DATA[#whichCase].threePhase := 0; END_IF;
   IF #_w1 THEN #whichCase := #whichCase + 1; END_IF;
END_REGION

REGION Network 5 (SCL): Automatyczna zmiana parametrów
   // Zmiana parametrów w zależności od aktualnego cyklu.
   #caseTime := DINT_TO_TIME(3*#I_switchTime);

   CASE #whichCase OF
       0:
           IF #I_start THEN
               #whichCase := 1;
           END_IF;

       1:
           #IO_power := 20;
           #IO_onePhase := FALSE;
           #IO_threePhase := TRUE;

       2:
           #IO_power := 50;
           #IO_onePhase := FALSE;
           #IO_threePhase := TRUE;

       3:
           #IO_power := 80;
           #IO_onePhase := FAlSE;
           #IO_threePhase := TRUE;

       4:
           #IO_power := 20;
           #IO_onePhase := TRUE;
           #IO_threePhase := FALSE;

       5:
           #IO_power := 50;
           #IO_onePhase := TRUE;
           #IO_threePhase := FALSE;

       6:
           #IO_power := 80;
           #IO_onePhase := TRUE;
           #IO_threePhase := FALSE;

       7:
           #IO_power := 0;
           #IO_onePhase := FALSE;
           #IO_threePhase := FALSE;
           #whichCase := 0;

   END_CASE;
END_REGION
END_FUNCTION_BLOCK

ORGANIZATION_BLOCK "Main"   // OB1, LAD, ProgramCycle
TITLE = "Main Program Sweep (Cycle)"
{ S7_Optimized_Access := 'TRUE' }
VERSION : 0.1
   VAR_INPUT
      Initial_Call : Bool;   // Initial call of this OB
      Remanence : Bool;   // =True, if remanent data are available
   END_VAR
   VAR_TEMP
      var : Variant;
      retval : Int;
   END_VAR
BEGIN

REGION Network 1: Wywołanie PWM
   // cycleTime - okres PWM (s)
   // switchTime - okres zmiany grzałek (s)
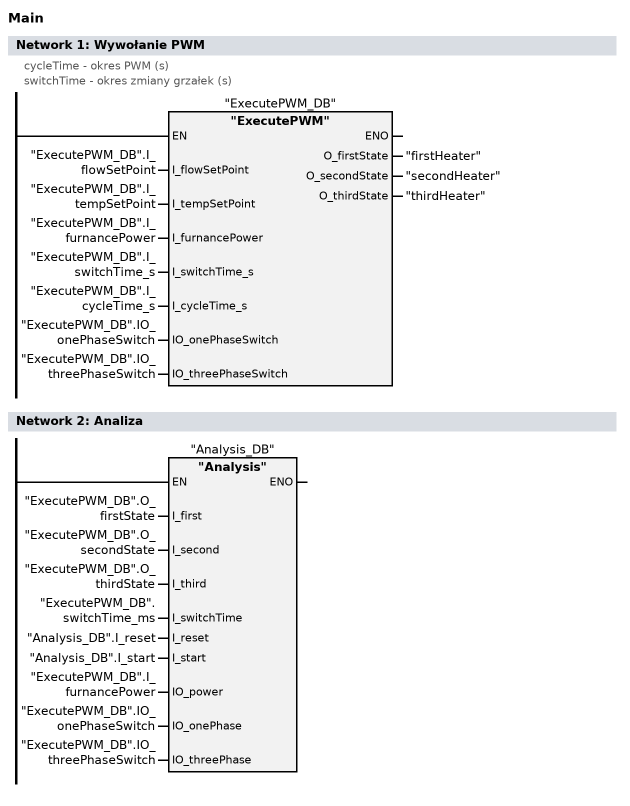
   RUNG wire#powerrail
      "ExecutePWM_DB"(I_flowSetPoint := "ExecutePWM_DB".I_flowSetPoint, I_tempSetPoint := "ExecutePWM_DB".I_tempSetPoint, I_furnancePower := "ExecutePWM_DB".I_furnancePower, I_switchTime_s := "ExecutePWM_DB".I_switchTime_s, I_cycleTime_s := "ExecutePWM_DB".I_cycleTime_s, IO_onePhaseSwitch := "ExecutePWM_DB".IO_onePhaseSwitch, IO_threePhaseSwitch := "ExecutePWM_DB".IO_threePhaseSwitch, O_firstState => "firstHeater", O_secondState => "secondHeater", O_thirdState => "thirdHeater")
   END_RUNG
   // the same network as SCL:
   "ExecutePWM_DB"(I_flowSetPoint := "ExecutePWM_DB".I_flowSetPoint,   // "ExecutePWM"
                   I_tempSetPoint := "ExecutePWM_DB".I_tempSetPoint,
                   I_furnancePower := "ExecutePWM_DB".I_furnancePower,
                   I_switchTime_s := "ExecutePWM_DB".I_switchTime_s,
                   I_cycleTime_s := "ExecutePWM_DB".I_cycleTime_s,
                   IO_onePhaseSwitch := "ExecutePWM_DB".IO_onePhaseSwitch,
                   IO_threePhaseSwitch := "ExecutePWM_DB".IO_threePhaseSwitch,
                   O_firstState => "firstHeater",
                   O_secondState => "secondHeater",
                   O_thirdState => "thirdHeater");
END_REGION

REGION Network 2: Analiza
   RUNG wire#powerrail
      "Analysis_DB"(I_first := "ExecutePWM_DB".O_firstState, I_second := "ExecutePWM_DB".O_secondState, I_third := "ExecutePWM_DB".O_thirdState, I_switchTime := "ExecutePWM_DB".switchTime_ms, I_reset := "Analysis_DB".I_reset, I_start := "Analysis_DB".I_start, IO_power := "ExecutePWM_DB".I_furnancePower, IO_onePhase := "ExecutePWM_DB".IO_onePhaseSwitch, IO_threePhase := "ExecutePWM_DB".IO_threePhaseSwitch)
   END_RUNG
   // the same network as SCL:
   "Analysis_DB"(I_first := "ExecutePWM_DB".O_firstState,   // "Analysis"
                 I_second := "ExecutePWM_DB".O_secondState,
                 I_third := "ExecutePWM_DB".O_thirdState,
                 I_switchTime := "ExecutePWM_DB".switchTime_ms,
                 I_reset := "Analysis_DB".I_reset,
                 I_start := "Analysis_DB".I_start,
                 IO_power := "ExecutePWM_DB".I_furnancePower,
                 IO_onePhase := "ExecutePWM_DB".IO_onePhaseSwitch,
                 IO_threePhase := "ExecutePWM_DB".IO_threePhaseSwitch);
END_REGION
END_ORGANIZATION_BLOCK

ORGANIZATION_BLOCK "Cyclic interrupt"   // OB30, LAD, CyclicInterrupt
{ S7_Optimized_Access := 'TRUE' }
VERSION : 0.1
   VAR_INPUT
      Initial_Call : Bool;   // Initial call of this OB
      Event_Count : Int;   // Events discarded
   END_VAR
BEGIN

REGION Network 1: Power PID
   // ...
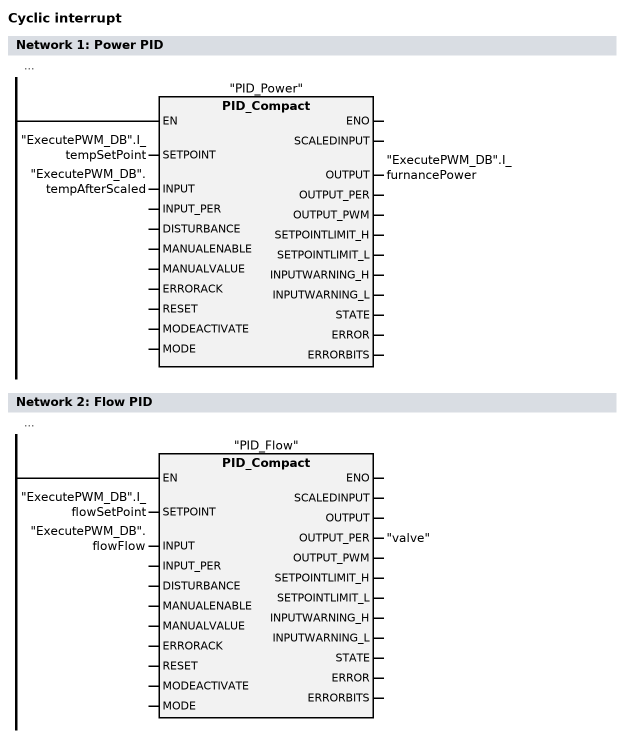
   "PID_Power"(Setpoint := "ExecutePWM_DB".I_tempSetPoint,   // PID_Compact
               Input := "ExecutePWM_DB".tempAfterScaled,
               Output => "ExecutePWM_DB".I_furnancePower);
END_REGION

REGION Network 2: Flow PID
   // ...
   "PID_Flow"(Setpoint := "ExecutePWM_DB".I_flowSetPoint,   // PID_Compact
              Input := "ExecutePWM_DB".flowFlow,
              Output_PER => "valve");
END_REGION
END_ORGANIZATION_BLOCK